Fanuc TP program (LS listing): mv_to_place.ls

/PROG  MV_TO_PLACE
/ATTR
DEFAULT_GROUP	= 1,*,*,*,*;
/MN
 : CALL MV_RETREAT ;
 :  ;
 : UFRAME_NUM=2 ;
 : UTOOL_NUM=2 ;
 : J PR[20:PLACE_PERCH] 100% CNT100 ;
/POS
/END
